(* IEC 61131-3 sources: moqui-plc/iec61131/moqui/framework/src/start, 10 files *)

(* ---- MoquiStartStatus.dut ---- *)
(*#-#-#-#-#-#-#-#-#-#---Declaration---#-#-#-#-#-#-#-#-#-#-#-#-#*)

{attribute 'qualified_only'}
{attribute 'strict'}
TYPE MoquiStartStatus : (
	Idle := 0,
	Run,
	Error
); END_TYPE

(* ---- MoquiStartStatus.st ---- *)
TYPE MoquiStartStatus : (
	Idle := 0,
	Run,
	Error
); END_TYPE

(* ---- LogDispatcher.pou ---- *)
(*#-#-#-#-#-#-#-#-#-#---Declaration---#-#-#-#-#-#-#-#-#-#-#-#-#*)

{attribute 'no_assign'}
PROGRAM LogDispatcher
VAR_EXTERNAL CONSTANT
    LOG_SOURCE_LIST_MAX_SIZE : UINT;
    LOG_MAX_SIZE : UINT;
	LOG_APPENDER_BATCH_SIZE : UINT;
END_VAR
VAR_EXTERNAL
    logSourceList : ARRAY[1..LOG_SOURCE_LIST_MAX_SIZE] OF LogSource;
    logSourceListSize : UINT;
    logAppenderEnable : BOOL;
END_VAR
VAR
    done, busy, error : BOOL;
    errorId : INT; (* 120 : LogSourceErr *)
    (* MQTT log appender *)
    logAppender : MqttLogAppender;
    currentSource : REFERENCE TO LogSource;
	currentLogBuffer : ARRAY[1..LOG_MAX_SIZE] OF LogEvent;
 	currentHead : UINT;
    currentTail : UINT;
    currentOverflowCount : UDINT;
    currentLogSize : UINT;
    sourceIndex : UINT := 1;
END_VAR

(*#-#-#-#-#-#-#-#-#-#---Implementation---#-#-#-#-#-#-#-#-#-#-#-#-#*)

IF NOT logAppenderEnable OR (logSourceListSize = 0) THEN
    done := FALSE; busy := FALSE; error := FALSE; errorId := 0;
    RETURN;
END_IF;

IF NOT logAppender.busy THEN
    IF sourceIndex < 1 OR sourceIndex > logSourceListSize THEN sourceIndex := 1; END_IF;

    currentSource REF= logSourceList[sourceIndex];
	(* Snapshot of the current metadata *)
	currentLogBuffer := currentSource.logRef.logBuffer;
    currentHead := currentSource.logRef.head;
    currentTail := currentSource.logRef.tail;
    currentOverflowCount := currentSource.logRef.overflowCount;
    currentLogSize := currentSource.logRef.logSize;

    (*
     * Skip this source if:
     *   - the buffer is empty, OR
     *   - fewer than LOG_APPENDER_BATCH_SIZE entries accumulated AND no overflow (no urgency).
     * Overflow bypasses the batch threshold to avoid losing entries.
     *)
    IF currentSource.logRef.isEmpty OR
            ((currentLogSize - currentSource.lastLogSize) < LOG_APPENDER_BATCH_SIZE) AND
             (currentOverflowCount <= currentSource.lastOverflowCount) THEN
        sourceIndex := (sourceIndex MOD logSourceListSize) + 1;
        RETURN;
    END_IF;

    (* Source ready: Commit snapshot metadata to LogSource *)
    currentSource.lastHead := currentHead;
    currentSource.lastTail := currentTail;
    currentSource.lastOverflowCount := currentOverflowCount;
    currentSource.lastLogSize := currentLogSize;
END_IF;

logAppender(execute := TRUE, logBuffer := currentLogBuffer, logBufferSize := currentLogSize,
	done => done, busy => busy, error => error, errorId => errorId);

IF logAppender.done OR logAppender.error THEN
    logAppender(execute := FALSE, done => done, busy => busy,
        error => error, errorId => errorId);
    (* Go to next log source *)
    sourceIndex := (sourceIndex MOD logSourceListSize) + 1;
END_IF;

(* ---- LogDispatcher.st ---- *)
PROGRAM LogDispatcher
	VAR_EXTERNAL CONSTANT
	    LOG_SOURCE_LIST_MAX_SIZE : UINT;
	    LOG_MAX_SIZE : UINT;
		LOG_APPENDER_BATCH_SIZE : UINT;
	END_VAR
	VAR_EXTERNAL
	    logSourceList : ARRAY[1..LOG_SOURCE_LIST_MAX_SIZE] OF LogSource;
	    logSourceListSize : UINT;
	    logAppenderEnable : BOOL;
	END_VAR
	VAR
	    done, busy, error : BOOL;
	    errorId : INT; (* 120 : LogSourceErr *)
	    (* MQTT log appender *)
	    logAppender : MqttLogAppender;
	    currentSource : REFERENCE TO LogSource;
		currentLogBuffer : ARRAY[1..LOG_MAX_SIZE] OF LogEvent;
	 	currentHead : UINT;
	    currentTail : UINT;
	    currentOverflowCount : UDINT;
	    currentLogSize : UINT;
	    sourceIndex : UINT := 1;
	END_VAR

	IF NOT logAppenderEnable OR (logSourceListSize = 0) THEN
	    done := FALSE; busy := FALSE; error := FALSE; errorId := 0;
	    RETURN;
	END_IF;

	IF NOT logAppender.busy THEN
	    IF sourceIndex < 1 OR sourceIndex > logSourceListSize THEN sourceIndex := 1; END_IF;

	    currentSource REF= logSourceList[sourceIndex];
		(* Snapshot of the current metadata *)
		currentLogBuffer := currentSource.logRef.logBuffer;
	    currentHead := currentSource.logRef.head;
	    currentTail := currentSource.logRef.tail;
	    currentOverflowCount := currentSource.logRef.overflowCount;
	    currentLogSize := currentSource.logRef.logSize;

	    (*
	     * Skip this source if:
	     *   - the buffer is empty, OR
	     *   - fewer than LOG_APPENDER_BATCH_SIZE entries accumulated AND no overflow (no urgency).
	     * Overflow bypasses the batch threshold to avoid losing entries.
	     *)
	    IF currentSource.logRef.isEmpty OR
	            ((currentLogSize - currentSource.lastLogSize) < LOG_APPENDER_BATCH_SIZE) AND
	             (currentOverflowCount <= currentSource.lastOverflowCount) THEN
	        sourceIndex := (sourceIndex MOD logSourceListSize) + 1;
	        RETURN;
	    END_IF;

	    (* Source ready: Commit snapshot metadata to LogSource *)
	    currentSource.lastHead := currentHead;
	    currentSource.lastTail := currentTail;
	    currentSource.lastOverflowCount := currentOverflowCount;
	    currentSource.lastLogSize := currentLogSize;
	END_IF;

	logAppender(execute := TRUE, logBuffer := currentLogBuffer, logBufferSize := currentLogSize,
		done => done, busy => busy, error => error, errorId => errorId);

	IF logAppender.done OR logAppender.error THEN
	    logAppender(execute := FALSE, done => done, busy => busy,
	        error => error, errorId => errorId);
	    (* Go to next log source *)
	    sourceIndex := (sourceIndex MOD logSourceListSize) + 1;
	END_IF;
	END_PROGRAM

(* ---- MoquiStart.pou ---- *)
(*#-#-#-#-#-#-#-#-#-#---Declaration---#-#-#-#-#-#-#-#-#-#-#-#-#*)

{attribute 'no_assign'}
PROGRAM MoquiStart
VAR_EXTERNAL CONSTANT
	retryOnError : BOOL;
	minRetryTime, maxRetryCount : UINT;
END_VAR
VAR_EXTERNAL
	clks : Clocks;
	enable, init, error, reset : BOOL;
	allConfigLoaded : BOOL;
	retryCount, retryTime : UINT;
END_VAR
VAR
	operationType : OperatingMode := OperatingMode.Init;
	status : MoquiStartStatus := MoquiStartStatus.Idle;
	(* Main framework components *)
	logger : LoggerFacade;
	runNetworkDgs : NetworkDiagnostics;
	clockGen : ClockGeneration;
	inputProcessing : InputSignalUpdate;
	outputProcessing : OutputSignalUpdate;
	(* Device config (recipe) management *)
	configMgmt : DeviceConfigMgmt;
	(* Application component *)
	main : Main;
	mainDone : BOOL;
END_VAR

(*#-#-#-#-#-#-#-#-#-#---Implementation---#-#-#-#-#-#-#-#-#-#-#-#-#*)

(* Set the operating mode *)
IF ec.init THEN
	(* Logger facade init *)
	logger.enable := TRUE; logger.loggerName := 'moqui';
	operationType := OperatingMode.Init;
ELSE
	operationType := OperatingMode.Run;
END_IF;

(* Timing generation *)
(*
 * Uncomment if you want to make loops shorter than 10 ms.
 * It is not recommended to go below 5 ms with the PLC.
 * The control loop (current) of the axes is in the servo drives.
 *)
(* clks.systemClock := NOT clks.systemClock; *)
clockGen(operationType := operationType);

(*
 * Always run internal procedures, timing generation, process inputs/outputs to ensure safe state
 * even in software error state, but not in case of hardware/firmware fault.
 *)
(* Run hardware fault detection procedures (run network and remote IO diagnostics). *)
runNetworkDgs(error => ec.error);
IF ec.error THEN
	(* Best if set by an external supervision system: init := FALSE; *)
	status := MoquiStartStatus.Idle;
	RETURN; (* Recycle until the fault condition disappears *)
END_IF;

(* Input virtualization *)
inputProcessing(operationType := operationType);

(* Start FMS *)
CASE status OF
    MoquiStartStatus.Idle :
		(* Waiting for error reset from supervision *)
        IF NOT ec.error AND ec.enable THEN
			logger(message := 'Framework started.', level := LogLevel.Info);
            mainDone := FALSE;
            status := MoquiStartStatus.Run;
        END_IF;

    MoquiStartStatus.Run :
        (* Device config (recipe) orchestration *)
        configMgmt(enable := ec.enable, configCompleted := mainDone,
            allConfigLoaded => allConfigLoaded, error => ec.error);

        IF configMgmt.error THEN
			status := MoquiStartStatus.Error;
        ELSIF NOT configMgmt.busy THEN
            IF allConfigLoaded THEN
				logger(message := 'All device configs loaded. Framework idle.', level := LogLevel.Info);
				(* Auto disable waiting for new device configs from Moqui or supervision *)
                ec.enable := FALSE;
                status := MoquiStartStatus.Idle;
			ELSE
                (*
                 * Run the component FSMs sequentially.
				 * The Main component can act as a dispatcher for invoking
                 * the system's FSM and its subsystems.
                 *)
                main(operationType := operationType, done => mainDone, error => ec.error);
				IF main.error THEN status := MoquiStartStatus.Error; END_IF;
            END_IF;
        END_IF;

    MoquiStartStatus.Error :
        (* Retry logic *)
		IF retryOnError AND (retryCount < maxRetryCount) THEN
			(* Retry timer update *)
			IF clks.clock1s THEN
				retryTime := retryTime + 1;
			END_IF;

			IF (retryTime >= minRetryTime) THEN
				logger(message := 'Retrying after error ...', level := LogLevel.Warn);
				retryCount := retryCount + 1;
				retryTime := 0; (* Reset the timer *)
				autoReset := TRUE; (* Auto reset *)
			END_IF;
		END_IF;

        IF reset OR autoReset THEN
            logger(message := 'Resetting framework after error.', level := LogLevel.Warn);
            ec.error := FALSE;
            retryCount := 0;
            retryTime := 0;
            status := MoquiStartStatus.Idle;
        END_IF;
END_CASE;

(* Output virtualization *)
outputProcessing(operationType := operationType);
(* Reset the init pulse *)
ec.init := FALSE;

(* ---- MoquiStart.st ---- *)
PROGRAM MoquiStart
	VAR_EXTERNAL CONSTANT
		retryOnError : BOOL;
		minRetryTime, maxRetryCount : UINT;
	END_VAR
	VAR_EXTERNAL
		clks : Clocks;
		enable, init, error, reset : BOOL;
		allConfigLoaded : BOOL;
		retryCount, retryTime : UINT;
	END_VAR
	VAR
		operationType : OperatingMode := OperatingMode.Init;
		status : MoquiStartStatus := MoquiStartStatus.Idle;
		(* Main framework components *)
		logger : LoggerFacade;
		runNetworkDgs : NetworkDiagnostics;
		clockGen : ClockGeneration;
		inputProcessing : InputSignalUpdate;
		outputProcessing : OutputSignalUpdate;
		(* Device config (recipe) management *)
		configMgmt : DeviceConfigMgmt;
		(* Application component *)
		main : Main;
		mainDone : BOOL;
		mainDoneREdge : R_TRIG;
		deviceConfigContextResetRequest : BOOL;
		(*
	     * Keep one Init cycle pending for Main after the first device config has
		 * been loaded, because recipe data also contains device init/homing params.
	     *)
		mainInitPending : BOOL := TRUE;
	END_VAR

	(* Set the operating mode *)
	IF ec.init THEN
		(* Logger facade init *)
		logger.enable := TRUE; logger.loggerName := 'moqui';
		operationType := OperatingMode.Init;
		mainInitPending := TRUE;
	ELSE
		operationType := OperatingMode.Run;
	END_IF;

	(* Timing generation *)
	(*
	 * Uncomment if you want to make loops shorter than 10 ms.
	 * It is not recommended to go below 5 ms with the PLC.
	 * The control loop (current) of the axes is in the servo drives.
	 *)
	(* clks.systemClock := NOT clks.systemClock; *)
	clockGen(operationType := operationType);

	(*
	 * Always run internal procedures, timing generation, process inputs/outputs to ensure safe state
	 * even in software error state, but not in case of hardware/firmware fault.
	 *)
	(* Run hardware fault detection procedures (run network and remote IO diagnostics). *)
	(* runNetworkDgs(error => ec.error);
	IF ec.error THEN
		(* Best if set by an external supervision system: init := FALSE; *)
		status := MoquiStartStatus.Idle;
		RETURN; (* Recycle until the fault condition disappears *)
	END_IF; *)

	(* Input virtualization *)
	(* inputProcessing(operationType := operationType); *)

	(*
	 * Device config (recipe) orchestration must also run during Init because the
	 * first recipe carries the device initialization and homing parameters.
	 *)
	configMgmt(enable := ec.enable, configCompleted := mainDone,
		allConfigLoaded => allConfigLoaded, error => ec.error);
	(*
	 * Main exposes completion as a level signal; derive a one-scan event here
	 * because recipe advancement and context reset are one-shot actions.
	 *)
	mainDoneREdge(CLK := mainDone);
	IF mainDoneREdge.Q THEN
		deviceConfigContextResetRequest := TRUE;
	END_IF;

	(* Start FMS *)
	CASE status OF
	    MoquiStartStatus.Idle :
			(* Waiting for error reset from supervision *)
	        IF NOT ec.error AND ec.enable THEN
				logger(message := 'Framework started.', level := LogLevel.Info);
	            mainDone := FALSE;
				deviceConfigContextResetRequest := FALSE;
	            status := MoquiStartStatus.Run;
	        END_IF;

	    MoquiStartStatus.Run :
	        IF configMgmt.error THEN
				status := MoquiStartStatus.Error;
	        ELSIF NOT configMgmt.busy THEN
	            IF allConfigLoaded THEN
					logger(message := 'All device configs loaded. Framework idle.', level := LogLevel.Info);
					(* Auto disable waiting for new device configs from Moqui or supervision *)
	                ec.enable := FALSE;
	                status := MoquiStartStatus.Idle;
				ELSE
	                (*
	                 * Run the component FSMs sequentially.
					 * The Main component can act as a dispatcher for invoking
	                 * the system's FSM and its subsystems.
					 *
					 * The very first call after recipe load must be Init so that
					 * all device FBs consume their recipe-based init/homing params.
	                 *)
	                main(operationType := SEL(mainInitPending, OperatingMode.Run, OperatingMode.Init),
						enable := ec.enable, deviceConfigContextResetRequest := deviceConfigContextResetRequest,
						done => mainDone, error => ec.error);
					mainInitPending := FALSE;
					deviceConfigContextResetRequest := FALSE;
					IF main.error THEN status := MoquiStartStatus.Error; END_IF;
	            END_IF;
	        END_IF;

	    MoquiStartStatus.Error :
	        (* Retry logic *)
			IF retryOnError AND (retryCount < maxRetryCount) THEN
				(* Retry timer update *)
				IF clks.clock1s THEN
					retryTime := retryTime + 1;
				END_IF;

				IF (retryTime >= minRetryTime) THEN
					logger(message := 'Retrying after error ...', level := LogLevel.Warn);
					retryCount := retryCount + 1;
					retryTime := 0; (* Reset the timer *)
					autoReset := TRUE; (* Auto reset *)
				END_IF;
			END_IF;

	        IF reset OR autoReset THEN
	            logger(message := 'Resetting framework after error.', level := LogLevel.Warn);
	            ec.error := FALSE;
	            retryCount := 0;
	            retryTime := 0;
				mainInitPending := TRUE;
				deviceConfigContextResetRequest := FALSE;
	            status := MoquiStartStatus.Idle;
	        END_IF;
	END_CASE;

	(* Output virtualization *)
	(* outputProcessing(operationType := operationType); *)
	(* Reset the init pulse *)
	ec.init := FALSE;
	END_PROGRAM

(* ---- MqttParameterPub.pou ---- *)
(*#-#-#-#-#-#-#-#-#-#---Declaration---#-#-#-#-#-#-#-#-#-#-#-#-#*)

{attribute 'no_assign'}
PROGRAM MqttParameterPub
VAR_EXTERNAL CONSTANT
	JSON_PAYLOAD_MAX_SIZE : UINT;
	pubPayloadFormatIndicator : BYTE;
	pubMessageExpiryInterval : UDINT;
	pubContentType : WSTRING(32);
	(* pubUserProperties : ARRAY [0..(MQTT.MQTTParam.g_udiMaxUserProperties - 1)] OF MQTT.MQTTStringPair; *)
	paramsPubQoS : MQTT.MQTT_QOS;
	paramsPubRetain : BOOL;
	paramsReDelivery : BOOL;
    liveParamsPubTopic : WSTRING(1024);
	liveParamsPubTimeout : UINT;
END_VAR
VAR_EXTERNAL
	paramsPubEnable : BOOL;
	connectionFactory : MqttConnectionFactory;
END_VAR
VAR
	done, busy, error : BOOL;
    errorId : INT;
	jsonPayload : WSTRING(JSON_PAYLOAD_MAX_SIZE);
	pubTopic : WSTRING(1024) := liveParamsPubTopic;
	pubMessage : STRING(JSON_PAYLOAD_MAX_SIZE);
	(* Publisher *)
	publisher : MQTT.MQTTPublish;
	(* Publish properties v5 *)
	mqttPublishProperties : MQTT.MQTTPublishProperties := (
		bPayloadFormatIndicator := pubPayloadFormatIndicator,
		wsContentType := pubContentType,
		udiMessageExpiryInterval := pubMessageExpiryInterval
		(* userProperties := pubUserProperties *)
	);
    (* JSON serializer *)
    parameterMapper : SerializeParametersToJson;
END_VAR

(*#-#-#-#-#-#-#-#-#-#---Implementation---#-#-#-#-#-#-#-#-#-#-#-#-#*)

(* Publishing disabled *)
IF NOT paramsPubEnable THEN
	done := FALSE; busy := FALSE; error := FALSE; errorId := 0;
	RETURN;
END_IF;

(* Connect to the broker *)
connectionFactory(connect := TRUE, error => error, errorId => errorId);
(* Reset and retry on next cycle *)
IF connectionFactory.connection.xError THEN
	connectionFactory(connect := FALSE, error => error, errorId => errorId);
	done := FALSE; busy := FALSE;
	RETURN;
END_IF;

(* Waiting for connection to broker *)
IF NOT connectionFactory.connected THEN RETURN; END_IF;

IF NOT publisher.xBusy THEN
	(* JSON mapping *)
	parameterMapper(execute := TRUE, jsonPayload => jsonPayload,
		busy => busy, error => error, errorId => errorId);
	IF parameterMapper.error THEN
		(* Reset JSON writer *)
		parameterMapper(execute := FALSE, error => error, errorId => errorId);
		done := FALSE; busy := FALSE;
		RETURN;
	END_IF;
END_IF;

IF parameterMapper.done THEN
	(* Publish the payload *)
	pubMessage := TO_STRING(jsonPayload);
	publisher(xExecute := TRUE, mqttClient := connectionFactory.connection, wsTopicName := pubTopic,
		pbPayload := ADR(pubMessage), udiPayloadSize := INT_TO_UDINT(LEN(pubMessage)),
		eQoS := paramsPubQoS, xReDelivery := paramsReDelivery, xRetain := paramsPubRetain,
		udiTimeOut := liveParamsPubTimeout, mQTTPublishProperties := mqttPublishProperties,
		xDone => done, xBusy => busy, xError => error, eMQTTError => errorId);

	IF publisher.xError OR publisher.xDone THEN
		(* Auto reset: next cycle restarts from scratch *)
		parameterMapper(execute := FALSE, busy => busy,
			error => error, errorId => errorId);
		publisher(xExecute := FALSE, mqttClient := connectionFactory.connection, wsTopicName := pubTopic,
			xDone => done, xBusy => busy, xError => error, eMQTTError => errorId);
	END_IF;
END_IF;

(* ---- MqttParameterPub.st ---- *)
PROGRAM MqttParameterPub
	VAR_EXTERNAL CONSTANT
		JSON_PAYLOAD_MAX_SIZE : UINT;
		pubPayloadFormatIndicator : BYTE;
		pubMessageExpiryInterval : UDINT;
		pubContentType : WSTRING(32);
		(* pubUserProperties : ARRAY [0..(MQTT.MQTTParam.g_udiMaxUserProperties - 1)] OF MQTT.MQTTStringPair; *)
		paramsPubQoS : MQTT.MQTT_QOS;
		paramsPubRetain : BOOL;
		paramsReDelivery : BOOL;
	    liveParamsPubTopic : WSTRING(1024);
		liveParamsPubTimeout : UINT;
	END_VAR
	VAR_EXTERNAL
		paramsPubEnable : BOOL;
		connectionFactory : MqttConnectionFactory;
	END_VAR
	VAR
		done, busy, error : BOOL;
	    errorId : INT;
		jsonPayload : WSTRING(JSON_PAYLOAD_MAX_SIZE);
		pubTopic : WSTRING(1024) := liveParamsPubTopic;
		pubMessage : STRING(JSON_PAYLOAD_MAX_SIZE);
		(* Publisher *)
		publisher : MQTT.MQTTPublish;
		(* Publish properties v5 *)
		mqttPublishProperties : MQTT.MQTTPublishProperties := (
			bPayloadFormatIndicator := pubPayloadFormatIndicator,
			wsContentType := pubContentType,
			udiMessageExpiryInterval := pubMessageExpiryInterval
			(* userProperties := pubUserProperties *)
		);
	    (* JSON serializer *)
	    parameterMapper : SerializeParametersToJson;
	END_VAR

	(* Publishing disabled *)
	IF NOT paramsPubEnable THEN
		done := FALSE; busy := FALSE; error := FALSE; errorId := 0;
		RETURN;
	END_IF;

	(* Connect to the broker *)
	connectionFactory(connect := TRUE, error => error, errorId => errorId);
	(* Reset and retry on next cycle *)
	IF connectionFactory.connection.xError THEN
		connectionFactory(connect := FALSE, error => error, errorId => errorId);
		done := FALSE; busy := FALSE;
		RETURN;
	END_IF;

	(* Waiting for connection to broker *)
	IF NOT connectionFactory.connected THEN RETURN; END_IF;

	IF NOT publisher.xBusy THEN
		(* JSON mapping *)
		parameterMapper(execute := TRUE, jsonPayload => jsonPayload,
			busy => busy, error => error, errorId => errorId);
		IF parameterMapper.error THEN
			(* Reset JSON writer *)
			parameterMapper(execute := FALSE, error => error, errorId => errorId);
			done := FALSE; busy := FALSE;
			RETURN;
		END_IF;
	END_IF;

	IF parameterMapper.done THEN
		(* Publish the payload *)
		pubMessage := TO_STRING(jsonPayload);
		publisher(xExecute := TRUE, mqttClient := connectionFactory.connection, wsTopicName := pubTopic,
			pbPayload := ADR(pubMessage), udiPayloadSize := INT_TO_UDINT(LEN(pubMessage)),
			eQoS := paramsPubQoS, xReDelivery := paramsReDelivery, xRetain := paramsPubRetain,
			udiTimeOut := liveParamsPubTimeout, mQTTPublishProperties := mqttPublishProperties,
			xDone => done, xBusy => busy, xError => error, eMQTTError => errorId);

		IF publisher.xError OR publisher.xDone THEN
			(* Auto reset: next cycle restarts from scratch *)
			parameterMapper(execute := FALSE, busy => busy,
				error => error, errorId => errorId);
			publisher(xExecute := FALSE, mqttClient := connectionFactory.connection, wsTopicName := pubTopic,
				xDone => done, xBusy => busy, xError => error, eMQTTError => errorId);
		END_IF;
	END_IF;
	END_PROGRAM

(* ---- MqttParameterSub.pou ---- *)
(*#-#-#-#-#-#-#-#-#-#---Declaration---#-#-#-#-#-#-#-#-#-#-#-#-#*)

{attribute 'no_assign'}
PROGRAM MqttParameterSub
VAR_EXTERNAL CONSTANT
	JSON_PAYLOAD_MAX_SIZE : UINT;
	(* Subscribe properties v5 *)
	subscriptionIdentifier : UDINT;
	(* subUserProperties : ARRAY [0..(MQTT.MQTTParam.g_udiMaxUserProperties - 1)] OF MQTT.MQTTStringPair; *)
	paramsSubQoS : MQTT.MQTT_QOS;
	paramsSubFilterMode : MQTT.FILTER_MODE;
	subNoLocalOption : BOOL;
	subRetainAsPublished : BOOL;
	subRetainHandling : MQTT.MQTT_RETAIN_HANDLING;
	liveParamsSubTopic : WSTRING(1024);
	liveParamsSubTimeout : UINT;
END_VAR
VAR_EXTERNAL
	paramsSubEnable : BOOL;
	connectionFactory : MqttConnectionFactory;
END_VAR
VAR
	done, busy, error : BOOL;
    errorId : INT;
	(* Subscriber *)
	subscriber : MQTT.MQTTSubscribe;
	(* Subscribe properties v5 *)
	mqttSubscribeProperties : MQTT.MQTTSubscribeProperties := (
		udiSubscriptionIdentifier := subscriptionIdentifier,
		xNoLocalOption := subNoLocalOption,
		xRetainAsPublished := subRetainAsPublished,
		eRetainHandling := subRetainHandling
		(* userProperties := subUserProperties; *)
	);
    (* JSON parser *)
    parser : DeserializeJsonToParameters;
	parserActive : BOOL; (* TRUE while parser is running across multiple cycles *)
	subTopicFilter : WSTRING(1024) := liveParamsSubTopic;
	(* Last incoming message *)
	lastSubMessage : STRING(JSON_PAYLOAD_MAX_SIZE);
    receivedPayload : WSTRING(JSON_PAYLOAD_MAX_SIZE);
	subscriberEnable : BOOL;
END_VAR

(*#-#-#-#-#-#-#-#-#-#---Implementation---#-#-#-#-#-#-#-#-#-#-#-#-#*)

(* Subscription disabled *)
IF NOT paramsSubEnable THEN
	done := FALSE; busy := FALSE; error := FALSE; errorId := 0;
    RETURN;
END_IF;

(* Connect to the broker *)
connectionFactory(connect := TRUE, error => error, errorId => errorId);
(* Reset and retry on next cycle *)
IF connectionFactory.connection.xError THEN
	connectionFactory(connect := FALSE, error => error, errorId => errorId);
	done := FALSE; busy := FALSE;
	RETURN;
END_IF;

(* Manage subscriber enable: disable for one cycle on error to reset the FB *)
IF subscriber.xError THEN
	subscriberEnable := FALSE;
ELSE
	subscriberEnable := connectionFactory.connected;
END_IF;

(* Drive subscriber continuously; xDone = subscription confirmed (sub ack), not end of session *)
subscriber(xEnable := subscriberEnable, mqttClient := connectionFactory.connection,
	eFilterMode := paramsSubFilterMode, wsTopicFilter := subTopicFilter, eSubscribeQoS := paramsSubQoS,
	udiTimeout := liveParamsSubTimeout, pbPayload := ADR(lastSubMessage),
	udiMaxPayloadSize := SIZEOF(lastSubMessage), mQTTSubscribeProperties := mqttSubscribeProperties,
	xDone => done, xBusy => busy, xError => error, eMQTTError => errorId);

(* xReceived pulses TRUE for one cycle only: latch parserActive to keep parser running *)
IF subscriber.xSubscribeActive AND subscriber.xReceived
		AND subscriber.wsLastTopic = subTopicFilter THEN
	receivedPayload := TO_WSTRING(lastSubMessage);
	parserActive := TRUE;
END_IF;

(* Drive parser every cycle until done/error, regardless of xReceived *)
IF parserActive THEN
	(* JSON parsing *)
	parser(execute := TRUE, jsonPayload := receivedPayload,
		busy => busy, error => error, errorId => errorId);

	IF parser.done OR parser.error THEN
		(* Auto reset: next cycle restarts from scratch *)
		parser(execute := FALSE, done => done, busy => busy,
			error => error, errorId => errorId);
		parserActive := FALSE;
	END_IF;
END_IF;

(* ---- MqttParameterSub.st ---- *)
PROGRAM MqttParameterSub
	VAR_EXTERNAL CONSTANT
		JSON_PAYLOAD_MAX_SIZE : UINT;
		(* Subscribe properties v5 *)
		subscriptionIdentifier : UDINT;
		(* subUserProperties : ARRAY [0..(MQTT.MQTTParam.g_udiMaxUserProperties - 1)] OF MQTT.MQTTStringPair; *)
		paramsSubQoS : MQTT.MQTT_QOS;
		paramsSubFilterMode : MQTT.FILTER_MODE;
		subNoLocalOption : BOOL;
		subRetainAsPublished : BOOL;
		subRetainHandling : MQTT.MQTT_RETAIN_HANDLING;
		liveParamsSubTopic : WSTRING(1024);
		liveParamsSubTimeout : UINT;
	END_VAR
	VAR_EXTERNAL
		paramsSubEnable : BOOL;
		connectionFactory : MqttConnectionFactory;
	END_VAR
	VAR
		done, busy, error : BOOL;
	    errorId : INT;
		(* Subscriber *)
		subscriber : MQTT.MQTTSubscribe;
		(* Subscribe properties v5 *)
		mqttSubscribeProperties : MQTT.MQTTSubscribeProperties := (
			udiSubscriptionIdentifier := subscriptionIdentifier,
			xNoLocalOption := subNoLocalOption,
			xRetainAsPublished := subRetainAsPublished,
			eRetainHandling := subRetainHandling
			(* userProperties := subUserProperties; *)
		);
	    (* JSON parser *)
	    parser : DeserializeJsonToParameters;
		parserActive : BOOL; (* TRUE while parser is running across multiple cycles *)
		subTopicFilter : WSTRING(1024) := liveParamsSubTopic;
		(* Last incoming message *)
		lastSubMessage : STRING(JSON_PAYLOAD_MAX_SIZE);
	    receivedPayload : WSTRING(JSON_PAYLOAD_MAX_SIZE);
		subscriberEnable : BOOL;
	END_VAR

	(* Subscription disabled *)
	IF NOT paramsSubEnable THEN
		done := FALSE; busy := FALSE; error := FALSE; errorId := 0;
	    RETURN;
	END_IF;

	(* Connect to the broker *)
	connectionFactory(connect := TRUE, error => error, errorId => errorId);
	(* Reset and retry on next cycle *)
	IF connectionFactory.connection.xError THEN
		connectionFactory(connect := FALSE, error => error, errorId => errorId);
		done := FALSE; busy := FALSE;
		RETURN;
	END_IF;

	(* Manage subscriber enable: disable for one cycle on error to reset the FB *)
	IF subscriber.xError THEN
		subscriberEnable := FALSE;
	ELSE
		subscriberEnable := connectionFactory.connected;
	END_IF;

	(* Drive subscriber continuously; xDone = subscription confirmed (sub ack), not end of session *)
	subscriber(xEnable := subscriberEnable, mqttClient := connectionFactory.connection,
		eFilterMode := paramsSubFilterMode, wsTopicFilter := subTopicFilter, eSubscribeQoS := paramsSubQoS,
		udiTimeout := liveParamsSubTimeout, pbPayload := ADR(lastSubMessage),
		udiMaxPayloadSize := SIZEOF(lastSubMessage), mQTTSubscribeProperties := mqttSubscribeProperties,
		xDone => done, xBusy => busy, xError => error, eMQTTError => errorId);

	(* xReceived pulses TRUE for one cycle only: latch parserActive to keep parser running *)
	IF subscriber.xSubscribeActive AND subscriber.xReceived
			AND subscriber.wsLastTopic = subTopicFilter THEN
		receivedPayload := TO_WSTRING(lastSubMessage);
		parserActive := TRUE;
	END_IF;

	(* Drive parser every cycle until done/error, regardless of xReceived *)
	IF parserActive THEN
		(* JSON parsing *)
		parser(execute := TRUE, jsonPayload := receivedPayload,
			busy => busy, error => error, errorId => errorId);

		IF parser.done OR parser.error THEN
			(* Auto reset: next cycle restarts from scratch *)
			parser(execute := FALSE, done => done, busy => busy,
				error => error, errorId => errorId);
			parserActive := FALSE;
		END_IF;
	END_IF;
	END_PROGRAM
